Staubli VAL3: strlength.pgx

public program strlength(string& pStr[], num pLen)
  local string lStrEmpty
  local string l_sTemp
begin
  lStrEmpty="                                        "
  // look for asian message
  if getDisplayLen(pStr)>pLen and pLen>0
    // need to divide the message
    if getDisplayLen(pStr)==len(pStr)
      if mid(pStr,1,pLen)!=" "
        // european message
        pStr=mid(pStr,pLen-1,0)
        pStr=pStr+"."
      else
        // found and empty space
        pStr=mid(pStr,pLen,0)
      endIf
    else
      // asian one
      call midPos(pStr,pLen,0,pStr)
    endIf
  else
    if getDisplayLen(pStr)<pLen
      // european
      if getDisplayLen(pStr)==len(pStr)
        pStr=pStr+mid(lStrEmpty,pLen-getDisplayLen(pStr),0)
      else
        // asian
        call midPos(lStrEmpty,pLen-getDisplayLen(pStr),0,l_sTemp)
        pStr=pStr+l_sTemp
      endIf
    else
      // they are the same
      //
    endIf
  endIf
end
